//	Function: ExtendLPIfPossible()
//	Description: Helper function
//				 Pass in a device that is controlled byt a SV - extend at low pressure if possible
//	Created by: Ben Hess
//	Created Date: June 27th, 2019

IF (__QUERYINTERFACE(device, extendLowPressureDevice)) THEN
	extendLowPressureDevice.ExtendLowPressure();
	ExtendLPIfPossible := TRUE;
ELSE
	ExtendLPIfPossible := FALSE;
END_IF

END_FUNCTION

// Testing/HelperFunctions/HomeIfNeeded
FUNCTION HomeIfNeeded : BOOL
VAR_INPUT
	Component : IComponent;
END_VAR
VAR
	homableDevice : IHomable;
END_VAR

//	Function: HomeIfNeeded()
//	Description: Helper function
//				 Pass in a component - if it has a homable motor, and is not yet homed, start homing
//	Created by: Ben Hess
//	Created Date: May 16th, 2019

IF (__QUERYINTERFACE(Component, homableDevice)) AND Component.OptionActive THEN
	IF homableDevice.IsHomed THEN
		HomeIfNeeded := TRUE;
		RETURN;
	ELSE
		homableDevice.HomeNow();
	END_IF
END_IF

END_FUNCTION

// Testing/HelperFunctions/MoveRequested
FUNCTION MoveRequested : BOOL
VAR_INPUT
	Component : IComponent;
END_VAR
VAR
	movableDevice : IPostHomeMove;
END_VAR

//	Function: MoveIfNeeded()
//	Description: Helper function
//				 Pass in a component - if it has a homable motor, and is not yet homed, start homing
//	Created by: Ben Hess
//	Created Date: May 16th, 2019

IF (__QUERYINTERFACE(Component, movableDevice)) AND Component.OptionActive THEN
	IF NOT movableDevice.InDesiredPosition THEN
		MoveRequested := TRUE;
		RETURN;
	ELSE
		RETURN;
	END_IF
END_IF

END_FUNCTION

// Testing/Motors/IPostHomeMove
INTERFACE IPostHomeMove

END_INTERFACE

// Testing/HelperFunctions/PostHomeMoveIfNeeded
FUNCTION PostHomeMoveIfNeeded : BOOL
VAR_INPUT
	Component : IComponent;
END_VAR
VAR
	movableDevice : IPostHomeMove;
END_VAR

//	Function: MoveIfNeeded()
//	Description: Helper function
//				 Pass in a component - if it has a homable motor, and is homed, and is configured for a post homing move, perform it
//	Created by: Ben Hess
//	Created Date: May 16th, 2019

IF (__QUERYINTERFACE(Component, movableDevice)) AND Component.OptionActive THEN
	IF movableDevice.InDesiredPosition THEN
		PostHomeMoveIfNeeded := TRUE;
		RETURN;
	ELSE
		movableDevice.MoveNow();
	END_IF
END_IF

END_FUNCTION

// Testing/Motors/FB_AppliedMotionMotor
FUNCTION_BLOCK FB_AppliedMotionMotor EXTENDS Axis_REF
VAR_INPUT
END_VAR
VAR_OUTPUT
END_VAR
VAR
END_VAR

END_FUNCTION_BLOCK

// UN00 - Sharp Bagger/EM01 - Bagger Head/TestBaggerHead
PROGRAM TestBaggerHead
VAR
END_VAR

END_PROGRAM

// /VISU_HELPER_Combobox_BagOpenFingersSelection
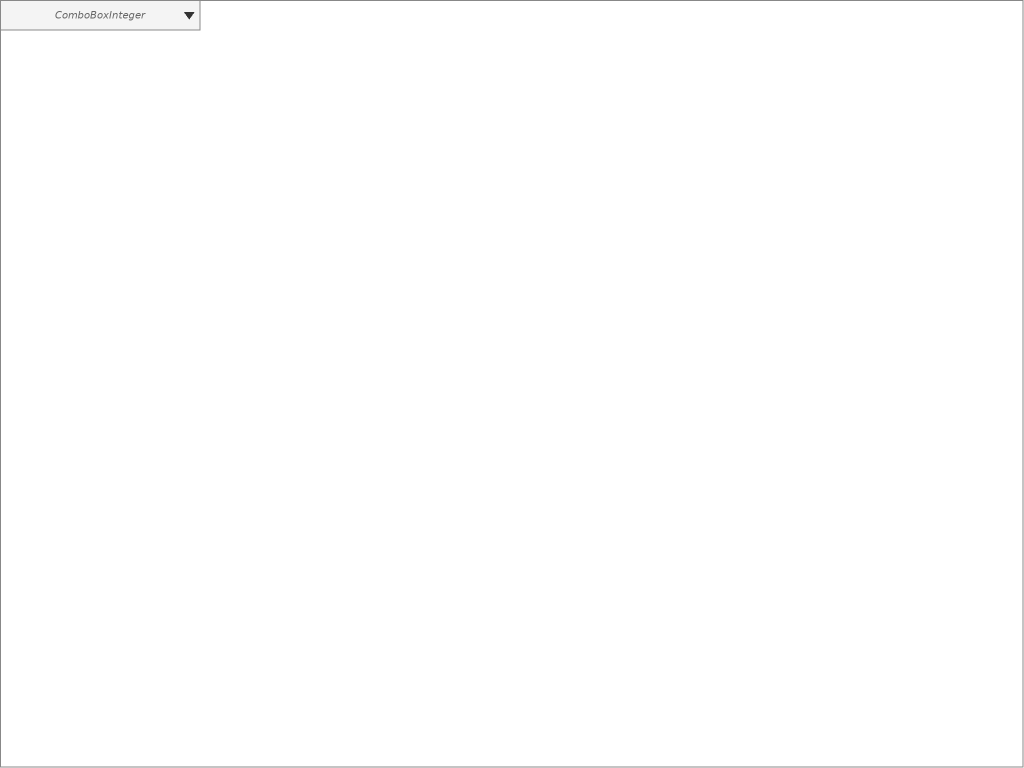
VISUALIZATION VISU_HELPER_Combobox_BagOpenFingersSelection  // 1024x768
VAR_IN_OUT
    varEnum : BagOpenFingersSelection;
END_VAR
    ComboBoxInteger (0,0 200x30), variable: varEnum, text list: 'TextListForCombobox_BagOpenFingersSelection'
END_VISUALIZATION

// /VISU_HELPER_Combobox_IntegratedConveyorSelection
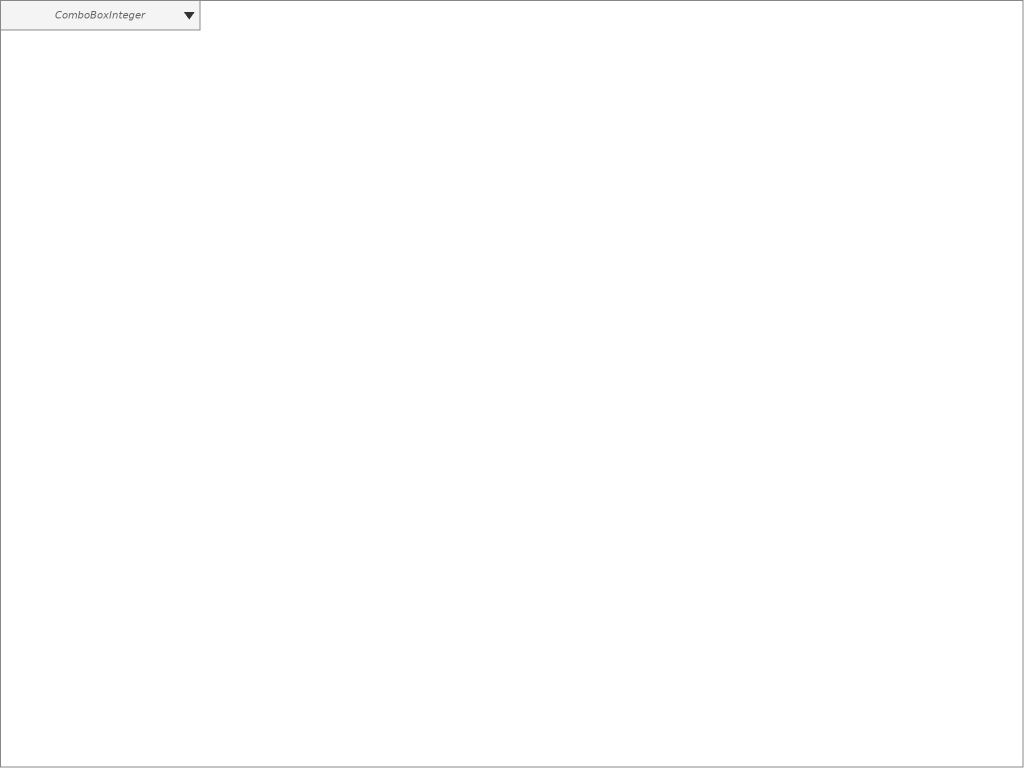
VISUALIZATION VISU_HELPER_Combobox_IntegratedConveyorSelection  // 1024x768
VAR_IN_OUT
    varEnum : IntegratedConveyorSelection;
END_VAR
    ComboBoxInteger (0,0 200x30), variable: varEnum, text list: 'TextListForCombobox_IntegratedConveyorSelection'
END_VISUALIZATION

// /VISU_HELPER_Combobox_LabelPrinterSelection
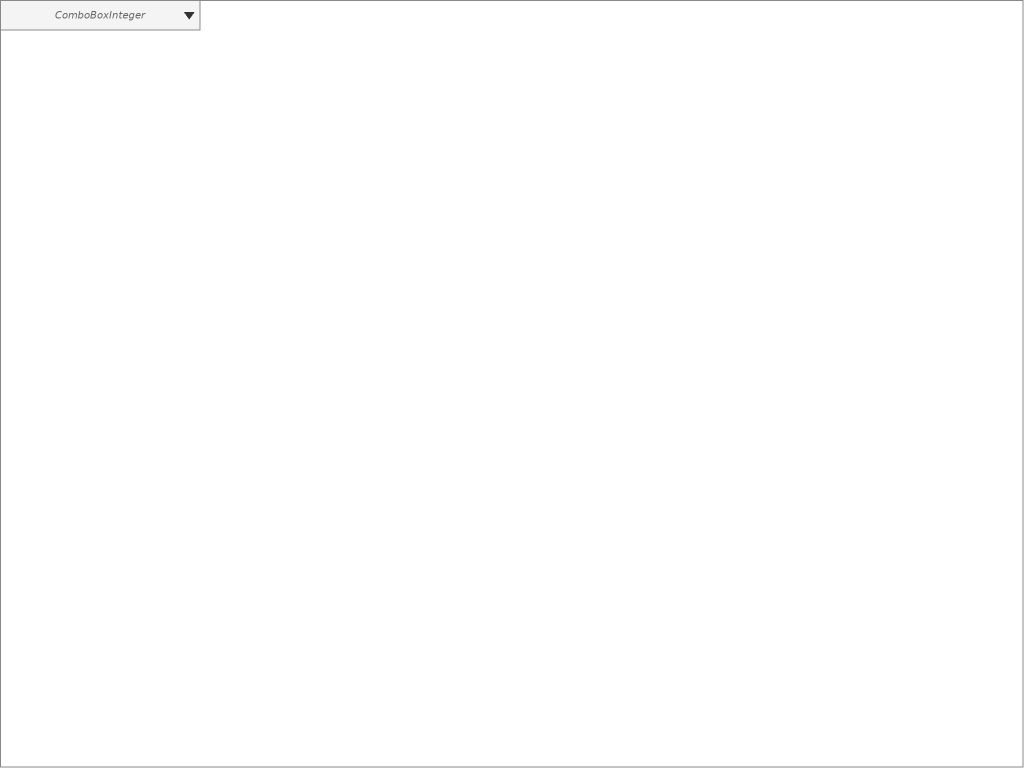
VISUALIZATION VISU_HELPER_Combobox_LabelPrinterSelection  // 1024x768
VAR_IN_OUT
    varEnum : LabelPrinterSelection;
END_VAR
    ComboBoxInteger (0,0 200x30), variable: varEnum, text list: 'TextListForCombobox_LabelPrinterSelection'
END_VISUALIZATION

// /VISU_HELPER_Combobox_PackageEjectionSelection
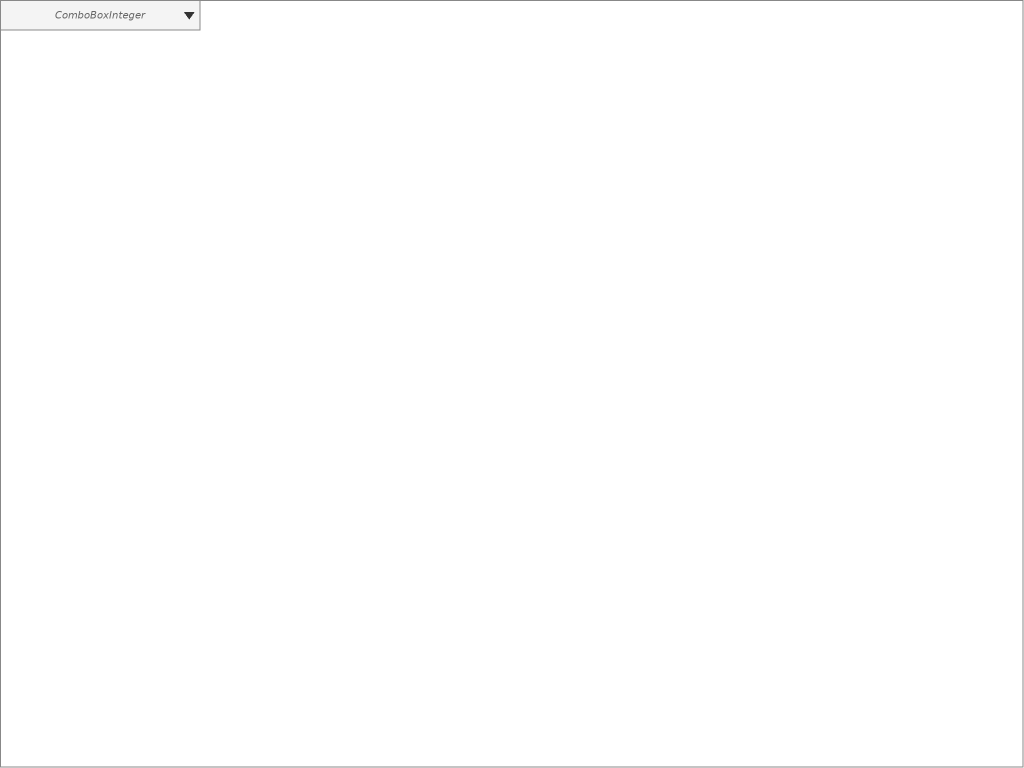
VISUALIZATION VISU_HELPER_Combobox_PackageEjectionSelection  // 1024x768
VAR_IN_OUT
    varEnum : PackageEjectionSelection;
END_VAR
    ComboBoxInteger (0,0 200x30), variable: varEnum, text list: 'TextListForCombobox_PackageEjectionSelection'
END_VISUALIZATION

// /VISU_HELPER_Combobox_SealFlattenerSelection
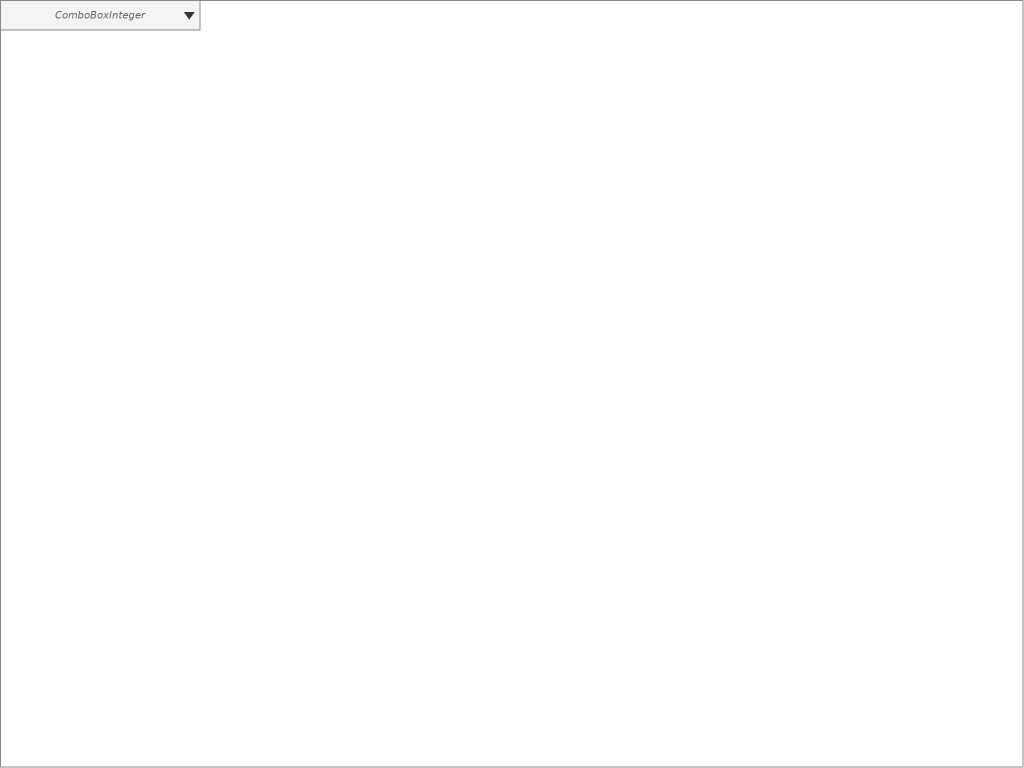
VISUALIZATION VISU_HELPER_Combobox_SealFlattenerSelection  // 1024x768
VAR_IN_OUT
    varEnum : SealFlattenerSelection;
END_VAR
    ComboBoxInteger (0,0 200x30), variable: varEnum, text list: 'TextListForCombobox_SealFlattenerSelection'
END_VISUALIZATION

// /VISU_NEW_FB_HMIData
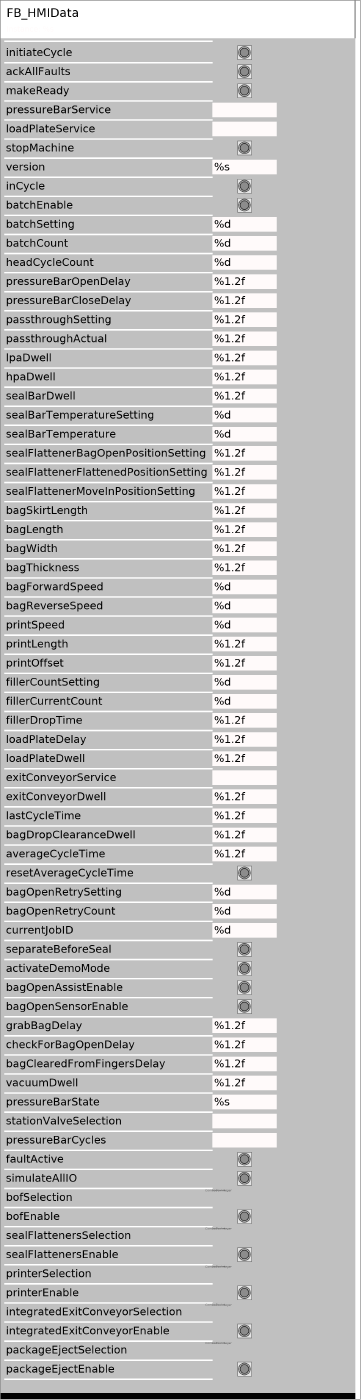
VISUALIZATION VISU_NEW_FB_HMIData  // 607x2348
VAR_INPUT
   {attribute 'parameterstringof' := 'm_Input_FB'}
   m_Input_INST_Str : STRING;
END_VAR
VAR_IN_OUT
   m_Input_FB : FB_HMIData;
END_VAR
    RoundedRectangle (0,0 597x81)
    RoundedRectangle (0,2306 597x40)
    Rectangle (0,64 597x2272)
    PushSwitch (399,76 24x24), variable: m_Input_FB.initiateCycle, behaviour: TOGGLE, style: Switch-PushSwitch-Gray
    PushSwitch (399,108 24x24), variable: m_Input_FB.ackAllFaults, behaviour: TOGGLE, style: Switch-PushSwitch-Gray
    PushSwitch (399,140 24x24), variable: m_Input_FB.makeReady, behaviour: TOGGLE, style: Switch-PushSwitch-Gray
    PushSwitch (399,236 24x24), variable: m_Input_FB.stopMachine, behaviour: TOGGLE, style: Switch-PushSwitch-Gray
    PushSwitch (399,300 24x24), variable: m_Input_FB.inCycle, behaviour: TOGGLE, style: Switch-PushSwitch-Gray
    PushSwitch (399,332 24x24), variable: m_Input_FB.batchEnable, behaviour: TOGGLE, style: Switch-PushSwitch-Gray
    PushSwitch (399,1452 24x24), variable: m_Input_FB.resetAverageCycleTime, behaviour: TOGGLE, style: Switch-PushSwitch-Gray
    PushSwitch (399,1580 24x24), variable: m_Input_FB.separateBeforeSeal, behaviour: TOGGLE, style: Switch-PushSwitch-Gray
    PushSwitch (399,1612 24x24), variable: m_Input_FB.activateDemoMode, behaviour: TOGGLE, style: Switch-PushSwitch-Gray
    PushSwitch (399,1644 24x24), variable: m_Input_FB.bagOpenAssistEnable, behaviour: TOGGLE, style: Switch-PushSwitch-Gray
    PushSwitch (399,1676 24x24), variable: m_Input_FB.bagOpenSensorEnable, behaviour: TOGGLE, style: Switch-PushSwitch-Gray
    PushSwitch (399,1932 24x24), variable: m_Input_FB.faultActive, behaviour: TOGGLE, style: Switch-PushSwitch-Gray
    PushSwitch (399,1964 24x24), variable: m_Input_FB.simulateAllIO, behaviour: TOGGLE, style: Switch-PushSwitch-Gray
    PushSwitch (399,2028 24x24), variable: m_Input_FB.bofEnable, behaviour: TOGGLE, style: Switch-PushSwitch-Gray
    PushSwitch (399,2092 24x24), variable: m_Input_FB.sealFlattenersEnable, behaviour: TOGGLE, style: Switch-PushSwitch-Gray
    PushSwitch (399,2156 24x24), variable: m_Input_FB.printerEnable, behaviour: TOGGLE, style: Switch-PushSwitch-Gray
    PushSwitch (399,2220 24x24), variable: m_Input_FB.integratedExitConveyorEnable, behaviour: TOGGLE, style: Switch-PushSwitch-Gray
    PushSwitch (399,2284 24x24), variable: m_Input_FB.packageEjectEnable, behaviour: TOGGLE, style: Switch-PushSwitch-Gray
    Rectangle (8,8 597x27), "FB_HMIData"
    Rectangle (8,35 597x27), "Instance: %s", text variable: m_Input_INST_Str
    Rectangle (7,68 350x2)
    Rectangle (7,76 350x24), "initiateCycle"
    Rectangle (7,104 350x2)
    Rectangle (7,108 350x24), "ackAllFaults"
    Rectangle (7,136 350x2)
    Rectangle (7,140 350x24), "makeReady"
    Rectangle (7,168 350x2)
    Rectangle (357,172 108x24), text variable: m_Input_FB.pressureBarService
        OnMouseClick: write the text variable via Default
    Rectangle (7,172 350x24), "pressureBarService"
    Rectangle (7,200 350x2)
    Rectangle (357,204 108x24), text variable: m_Input_FB.loadPlateService
        OnMouseClick: write the text variable via Default
    Rectangle (7,204 350x24), "loadPlateService"
    Rectangle (7,232 350x2)
    Rectangle (7,236 350x24), "stopMachine"
    Rectangle (7,264 350x2)
    Rectangle (357,268 108x24), "%s", text variable: m_Input_FB.version
        OnMouseClick: write the text variable via Default
    Rectangle (7,268 350x24), "version"
    Rectangle (7,296 350x2)
    Rectangle (7,300 350x24), "inCycle"
    Rectangle (7,328 350x2)
    Rectangle (7,332 350x24), "batchEnable"
    Rectangle (7,360 350x2)
    Rectangle (357,364 108x24), "%d", text variable: m_Input_FB.batchSetting
        OnMouseClick: write the text variable via Default
    Rectangle (7,364 350x24), "batchSetting"
    Rectangle (7,392 350x2)
    Rectangle (357,396 108x24), "%d", text variable: m_Input_FB.batchCount
        OnMouseClick: write the text variable via Default
    Rectangle (7,396 350x24), "batchCount"
    Rectangle (7,424 350x2)
    Rectangle (357,428 108x24), "%d", text variable: m_Input_FB.headCycleCount
        OnMouseClick: write the text variable via Default
    Rectangle (7,428 350x24), "headCycleCount"
    Rectangle (7,456 350x2)
    Rectangle (357,460 108x24), "%1.2f", text variable: m_Input_FB.pressureBarOpenDelay
        OnMouseClick: write the text variable via Default
    Rectangle (7,460 350x24), "pressureBarOpenDelay"
    Rectangle (7,488 350x2)
    Rectangle (357,492 108x24), "%1.2f", text variable: m_Input_FB.pressureBarCloseDelay
        OnMouseClick: write the text variable via Default
    Rectangle (7,492 350x24), "pressureBarCloseDelay"
    Rectangle (7,520 350x2)
    Rectangle (357,524 108x24), "%1.2f", text variable: m_Input_FB.passthroughSetting
        OnMouseClick: write the text variable via Default
    Rectangle (7,524 350x24), "passthroughSetting"
    Rectangle (7,552 350x2)
    Rectangle (357,556 108x24), "%1.2f", text variable: m_Input_FB.passthroughActual
        OnMouseClick: write the text variable via Default
    Rectangle (7,556 350x24), "passthroughActual"
    Rectangle (7,584 350x2)
    Rectangle (357,588 108x24), "%1.2f", text variable: m_Input_FB.lpaDwell
        OnMouseClick: write the text variable via Default
    Rectangle (7,588 350x24), "lpaDwell"
    Rectangle (7,616 350x2)
    Rectangle (357,620 108x24), "%1.2f", text variable: m_Input_FB.hpaDwell
        OnMouseClick: write the text variable via Default
    Rectangle (7,620 350x24), "hpaDwell"
    Rectangle (7,648 350x2)
    Rectangle (357,652 108x24), "%1.2f", text variable: m_Input_FB.sealBarDwell
        OnMouseClick: write the text variable via Default
    Rectangle (7,652 350x24), "sealBarDwell"
    Rectangle (7,680 350x2)
    Rectangle (357,684 108x24), "%d", text variable: m_Input_FB.sealBarTemperatureSetting
        OnMouseClick: write the text variable via Default
    Rectangle (7,684 350x24), "sealBarTemperatureSetting"
    Rectangle (7,712 350x2)
    Rectangle (357,716 108x24), "%d", text variable: m_Input_FB.sealBarTemperature
        OnMouseClick: write the text variable via Default
    Rectangle (7,716 350x24), "sealBarTemperature"
    Rectangle (7,744 350x2)
    Rectangle (357,748 108x24), "%1.2f", text variable: m_Input_FB.sealFlattenerBagOpenPositionSetting
        OnMouseClick: write the text variable via Default
    Rectangle (7,748 350x24), "sealFlattenerBagOpenPositionSetting"
    Rectangle (7,776 350x2)
    Rectangle (357,780 108x24), "%1.2f", text variable: m_Input_FB.sealFlattenerFlattenedPositionSetting
        OnMouseClick: write the text variable via Default
    Rectangle (7,780 350x24), "sealFlattenerFlattenedPositionSetting"
    Rectangle (7,808 350x2)
    Rectangle (357,812 108x24), "%1.2f", text variable: m_Input_FB.sealFlattenerMoveInPositionSetting
        OnMouseClick: write the text variable via Default
    Rectangle (7,812 350x24), "sealFlattenerMoveInPositionSetting"
    Rectangle (7,840 350x2)
    Rectangle (357,844 108x24), "%1.2f", text variable: m_Input_FB.bagSkirtLength
        OnMouseClick: write the text variable via Default
    Rectangle (7,844 350x24), "bagSkirtLength"
    Rectangle (7,872 350x2)
    Rectangle (357,876 108x24), "%1.2f", text variable: m_Input_FB.bagLength
        OnMouseClick: write the text variable via Default
    Rectangle (7,876 350x24), "bagLength"
    Rectangle (7,904 350x2)
    Rectangle (357,908 108x24), "%1.2f", text variable: m_Input_FB.bagWidth
        OnMouseClick: write the text variable via Default
    Rectangle (7,908 350x24), "bagWidth"
    Rectangle (7,936 350x2)
    Rectangle (357,940 108x24), "%1.2f", text variable: m_Input_FB.bagThickness
        OnMouseClick: write the text variable via Default
    Rectangle (7,940 350x24), "bagThickness"
    Rectangle (7,968 350x2)
    Rectangle (357,972 108x24), "%d", text variable: m_Input_FB.bagForwardSpeed
        OnMouseClick: write the text variable via Default
    Rectangle (7,972 350x24), "bagForwardSpeed"
    Rectangle (7,1000 350x2)
    Rectangle (357,1004 108x24), "%d", text variable: m_Input_FB.bagReverseSpeed
        OnMouseClick: write the text variable via Default
    Rectangle (7,1004 350x24), "bagReverseSpeed"
    Rectangle (7,1032 350x2)
    Rectangle (357,1036 108x24), "%d", text variable: m_Input_FB.printSpeed
        OnMouseClick: write the text variable via Default
    Rectangle (7,1036 350x24), "printSpeed"
    Rectangle (7,1064 350x2)
    Rectangle (357,1068 108x24), "%1.2f", text variable: m_Input_FB.printLength
        OnMouseClick: write the text variable via Default
    Rectangle (7,1068 350x24), "printLength"
    Rectangle (7,1096 350x2)
    Rectangle (357,1100 108x24), "%1.2f", text variable: m_Input_FB.printOffset
        OnMouseClick: write the text variable via Default
    Rectangle (7,1100 350x24), "printOffset"
    Rectangle (7,1128 350x2)
    Rectangle (357,1132 108x24), "%d", text variable: m_Input_FB.fillerCountSetting
        OnMouseClick: write the text variable via Default
    Rectangle (7,1132 350x24), "fillerCountSetting"
    Rectangle (7,1160 350x2)
    Rectangle (357,1164 108x24), "%d", text variable: m_Input_FB.fillerCurrentCount
        OnMouseClick: write the text variable via Default
    Rectangle (7,1164 350x24), "fillerCurrentCount"
    Rectangle (7,1192 350x2)
    Rectangle (357,1196 108x24), "%1.2f", text variable: m_Input_FB.fillerDropTime
        OnMouseClick: write the text variable via Default
    Rectangle (7,1196 350x24), "fillerDropTime"
    Rectangle (7,1224 350x2)
    Rectangle (357,1228 108x24), "%1.2f", text variable: m_Input_FB.loadPlateDelay
        OnMouseClick: write the text variable via Default
    Rectangle (7,1228 350x24), "loadPlateDelay"
    Rectangle (7,1256 350x2)
    Rectangle (357,1260 108x24), "%1.2f", text variable: m_Input_FB.loadPlateDwell
        OnMouseClick: write the text variable via Default
    Rectangle (7,1260 350x24), "loadPlateDwell"
    Rectangle (7,1288 350x2)
    Rectangle (357,1292 108x24), text variable: m_Input_FB.exitConveyorService
        OnMouseClick: write the text variable via Default
    Rectangle (7,1292 350x24), "exitConveyorService"
    Rectangle (7,1320 350x2)
    Rectangle (357,1324 108x24), "%1.2f", text variable: m_Input_FB.exitConveyorDwell
        OnMouseClick: write the text variable via Default
    Rectangle (7,1324 350x24), "exitConveyorDwell"
    Rectangle (7,1352 350x2)
    Rectangle (357,1356 108x24), "%1.2f", text variable: m_Input_FB.lastCycleTime
        OnMouseClick: write the text variable via Default
    Rectangle (7,1356 350x24), "lastCycleTime"
    Rectangle (7,1384 350x2)
    Rectangle (357,1388 108x24), "%1.2f", text variable: m_Input_FB.bagDropClearanceDwell
        OnMouseClick: write the text variable via Default
    Rectangle (7,1388 350x24), "bagDropClearanceDwell"
    Rectangle (7,1416 350x2)
    Rectangle (357,1420 108x24), "%1.2f", text variable: m_Input_FB.averageCycleTime
        OnMouseClick: write the text variable via Default
    Rectangle (7,1420 350x24), "averageCycleTime"
    Rectangle (7,1448 350x2)
    Rectangle (7,1452 350x24), "resetAverageCycleTime"
    Rectangle (7,1480 350x2)
    Rectangle (357,1484 108x24), "%d", text variable: m_Input_FB.bagOpenRetrySetting
        OnMouseClick: write the text variable via Default
    Rectangle (7,1484 350x24), "bagOpenRetrySetting"
    Rectangle (7,1512 350x2)
    Rectangle (357,1516 108x24), "%d", text variable: m_Input_FB.bagOpenRetryCount
        OnMouseClick: write the text variable via Default
    Rectangle (7,1516 350x24), "bagOpenRetryCount"
    Rectangle (7,1544 350x2)
    Rectangle (357,1548 108x24), "%d", text variable: m_Input_FB.currentJobID
        OnMouseClick: write the text variable via Default
    Rectangle (7,1548 350x24), "currentJobID"
    Rectangle (7,1576 350x2)
    Rectangle (7,1580 350x24), "separateBeforeSeal"
    Rectangle (7,1608 350x2)
    Rectangle (7,1612 350x24), "activateDemoMode"
    Rectangle (7,1640 350x2)
    Rectangle (7,1644 350x24), "bagOpenAssistEnable"
    Rectangle (7,1672 350x2)
    Rectangle (7,1676 350x24), "bagOpenSensorEnable"
    Rectangle (7,1704 350x2)
    Rectangle (357,1708 108x24), "%1.2f", text variable: m_Input_FB.grabBagDelay
        OnMouseClick: write the text variable via Default
    Rectangle (7,1708 350x24), "grabBagDelay"
    Rectangle (7,1736 350x2)
    Rectangle (357,1740 108x24), "%1.2f", text variable: m_Input_FB.checkForBagOpenDelay
        OnMouseClick: write the text variable via Default
    Rectangle (7,1740 350x24), "checkForBagOpenDelay"
    Rectangle (7,1768 350x2)
    Rectangle (357,1772 108x24), "%1.2f", text variable: m_Input_FB.bagClearedFromFingersDelay
        OnMouseClick: write the text variable via Default
    Rectangle (7,1772 350x24), "bagClearedFromFingersDelay"
    Rectangle (7,1800 350x2)
    Rectangle (357,1804 108x24), "%1.2f", text variable: m_Input_FB.vacuumDwell
        OnMouseClick: write the text variable via Default
    Rectangle (7,1804 350x24), "vacuumDwell"
    Rectangle (7,1832 350x2)
    Rectangle (357,1836 108x24), "%s", text variable: m_Input_FB.pressureBarState
        OnMouseClick: write the text variable via Default
    Rectangle (7,1836 350x24), "pressureBarState"
    Rectangle (7,1864 350x2)
    Rectangle (357,1868 108x24), text variable: m_Input_FB.stationValveSelection
        OnMouseClick: write the text variable via Default
    Rectangle (7,1868 350x24), "stationValveSelection"
    Rectangle (7,1896 350x2)
    Rectangle (357,1900 108x24), text variable: m_Input_FB.pressureBarCycles
        OnMouseClick: write the text variable via Default
    Rectangle (7,1900 350x24), "pressureBarCycles"
    Rectangle (7,1928 350x2)
    Rectangle (7,1932 350x24), "faultActive"
    Rectangle (7,1960 350x2)
    Rectangle (7,1964 350x24), "simulateAllIO"
    Rectangle (7,1992 350x2)
    Rectangle (7,1996 350x24), "bofSelection"
    Rectangle (7,2024 350x2)
    Rectangle (7,2028 350x24), "bofEnable"
    Rectangle (7,2056 350x2)
    Rectangle (7,2060 350x24), "sealFlattenersSelection"
    Rectangle (7,2088 350x2)
    Rectangle (7,2092 350x24), "sealFlattenersEnable"
    Rectangle (7,2120 350x2)
    Rectangle (7,2124 350x24), "printerSelection"
    Rectangle (7,2152 350x2)
    Rectangle (7,2156 350x24), "printerEnable"
    Rectangle (7,2184 350x2)
    Rectangle (7,2188 350x24), "integratedExitConveyorSelection"
    Rectangle (7,2216 350x2)
    Rectangle (7,2220 350x24), "integratedExitConveyorEnable"
    Rectangle (7,2248 350x2)
    Rectangle (7,2252 350x24), "packageEjectSelection"
    Rectangle (7,2280 350x2)
    Rectangle (7,2284 350x24), "packageEjectEnable"
    Rectangle (7,2312 350x2)
    Frame (357,1996 108x24)
        shows VISU_HELPER_Combobox_BagOpenFingersSelection(varEnum := m_Input_FB.bofSelection)
    Frame (357,2060 108x24)
        shows VISU_HELPER_Combobox_SealFlattenerSelection(varEnum := m_Input_FB.sealFlattenersSelection)
    Frame (357,2124 108x24)
        shows VISU_HELPER_Combobox_LabelPrinterSelection(varEnum := m_Input_FB.printerSelection)
    Frame (357,2188 108x24)
        shows VISU_HELPER_Combobox_IntegratedConveyorSelection(varEnum := m_Input_FB.integratedExitConveyorSelection)
    Frame (357,2252 108x24)
        shows VISU_HELPER_Combobox_PackageEjectionSelection(varEnum := m_Input_FB.packageEjectSelection)
END_VISUALIZATION

// /VISU_NEW_FB_IOLinkBlock
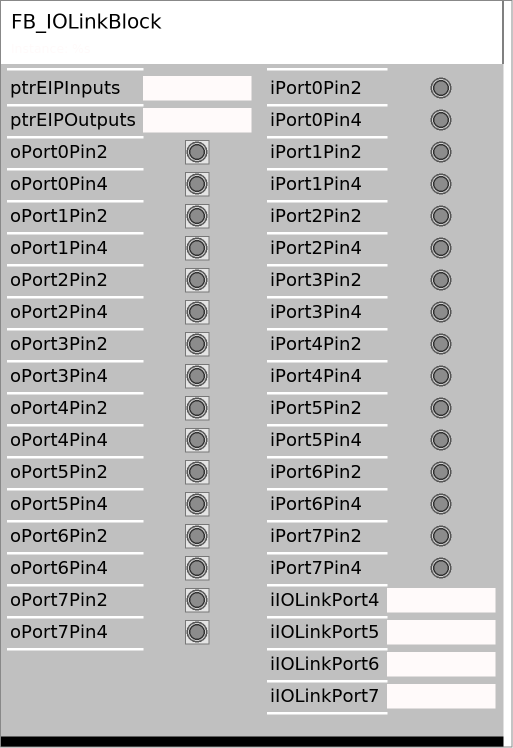
VISUALIZATION VISU_NEW_FB_IOLinkBlock  // 513x748
VAR_INPUT
   {attribute 'parameterstringof' := 'm_Input_FB'}
   m_Input_INST_Str : STRING;
END_VAR
VAR_IN_OUT
   m_Input_FB : FB_IOLinkBlock;
END_VAR
    RoundedRectangle (0,0 503x81)
    RoundedRectangle (0,706 503x40)
    Rectangle (0,64 503x672)
    Lamp1 (429,76 24x24), variable: m_Input_FB.iPort0Pin2, style: Lamp-Lamp1-Gray
    Lamp1 (429,108 24x24), variable: m_Input_FB.iPort0Pin4, style: Lamp-Lamp1-Gray
    Lamp1 (429,140 24x24), variable: m_Input_FB.iPort1Pin2, style: Lamp-Lamp1-Gray
    Lamp1 (429,172 24x24), variable: m_Input_FB.iPort1Pin4, style: Lamp-Lamp1-Gray
    Lamp1 (429,204 24x24), variable: m_Input_FB.iPort2Pin2, style: Lamp-Lamp1-Gray
    Lamp1 (429,236 24x24), variable: m_Input_FB.iPort2Pin4, style: Lamp-Lamp1-Gray
    Lamp1 (429,268 24x24), variable: m_Input_FB.iPort3Pin2, style: Lamp-Lamp1-Gray
    Lamp1 (429,300 24x24), variable: m_Input_FB.iPort3Pin4, style: Lamp-Lamp1-Gray
    Lamp1 (429,332 24x24), variable: m_Input_FB.iPort4Pin2, style: Lamp-Lamp1-Gray
    Lamp1 (429,364 24x24), variable: m_Input_FB.iPort4Pin4, style: Lamp-Lamp1-Gray
    Lamp1 (429,396 24x24), variable: m_Input_FB.iPort5Pin2, style: Lamp-Lamp1-Gray
    Lamp1 (429,428 24x24), variable: m_Input_FB.iPort5Pin4, style: Lamp-Lamp1-Gray
    Lamp1 (429,460 24x24), variable: m_Input_FB.iPort6Pin2, style: Lamp-Lamp1-Gray
    Lamp1 (429,492 24x24), variable: m_Input_FB.iPort6Pin4, style: Lamp-Lamp1-Gray
    Lamp1 (429,524 24x24), variable: m_Input_FB.iPort7Pin2, style: Lamp-Lamp1-Gray
    Lamp1 (429,556 24x24), variable: m_Input_FB.iPort7Pin4, style: Lamp-Lamp1-Gray
    PushSwitch (185,140 24x24), variable: m_Input_FB.oPort0Pin2, behaviour: TOGGLE, style: Switch-PushSwitch-Gray
    PushSwitch (185,172 24x24), variable: m_Input_FB.oPort0Pin4, behaviour: TOGGLE, style: Switch-PushSwitch-Gray
    PushSwitch (185,204 24x24), variable: m_Input_FB.oPort1Pin2, behaviour: TOGGLE, style: Switch-PushSwitch-Gray
    PushSwitch (185,236 24x24), variable: m_Input_FB.oPort1Pin4, behaviour: TOGGLE, style: Switch-PushSwitch-Gray
    PushSwitch (185,268 24x24), variable: m_Input_FB.oPort2Pin2, behaviour: TOGGLE, style: Switch-PushSwitch-Gray
    PushSwitch (185,300 24x24), variable: m_Input_FB.oPort2Pin4, behaviour: TOGGLE, style: Switch-PushSwitch-Gray
    PushSwitch (185,332 24x24), variable: m_Input_FB.oPort3Pin2, behaviour: TOGGLE, style: Switch-PushSwitch-Gray
    PushSwitch (185,364 24x24), variable: m_Input_FB.oPort3Pin4, behaviour: TOGGLE, style: Switch-PushSwitch-Gray
    PushSwitch (185,396 24x24), variable: m_Input_FB.oPort4Pin2, behaviour: TOGGLE, style: Switch-PushSwitch-Gray
    PushSwitch (185,428 24x24), variable: m_Input_FB.oPort4Pin4, behaviour: TOGGLE, style: Switch-PushSwitch-Gray
    PushSwitch (185,460 24x24), variable: m_Input_FB.oPort5Pin2, behaviour: TOGGLE, style: Switch-PushSwitch-Gray
    PushSwitch (185,492 24x24), variable: m_Input_FB.oPort5Pin4, behaviour: TOGGLE, style: Switch-PushSwitch-Gray
    PushSwitch (185,524 24x24), variable: m_Input_FB.oPort6Pin2, behaviour: TOGGLE, style: Switch-PushSwitch-Gray
    PushSwitch (185,556 24x24), variable: m_Input_FB.oPort6Pin4, behaviour: TOGGLE, style: Switch-PushSwitch-Gray
    PushSwitch (185,588 24x24), variable: m_Input_FB.oPort7Pin2, behaviour: TOGGLE, style: Switch-PushSwitch-Gray
    PushSwitch (185,620 24x24), variable: m_Input_FB.oPort7Pin4, behaviour: TOGGLE, style: Switch-PushSwitch-Gray
    Rectangle (8,8 503x27), "FB_IOLinkBlock"
    Rectangle (8,35 503x27), "Instance: %s", text variable: m_Input_INST_Str
    Rectangle (7,68 136x2)
    Rectangle (143,76 108x24), text variable: m_Input_FB.ptrEIPInputs
        OnMouseClick: write the text variable via Default
    Rectangle (7,76 136x24), "ptrEIPInputs"
    Rectangle (7,104 136x2)
    Rectangle (143,108 108x24), text variable: m_Input_FB.ptrEIPOutputs
        OnMouseClick: write the text variable via Default
    Rectangle (7,108 136x24), "ptrEIPOutputs"
    Rectangle (7,136 136x2)
    Rectangle (7,140 136x24), "oPort0Pin2"
    Rectangle (7,168 136x2)
    Rectangle (7,172 136x24), "oPort0Pin4"
    Rectangle (7,200 136x2)
    Rectangle (7,204 136x24), "oPort1Pin2"
    Rectangle (7,232 136x2)
    Rectangle (7,236 136x24), "oPort1Pin4"
    Rectangle (7,264 136x2)
    Rectangle (7,268 136x24), "oPort2Pin2"
    Rectangle (7,296 136x2)
    Rectangle (7,300 136x24), "oPort2Pin4"
    Rectangle (7,328 136x2)
    Rectangle (7,332 136x24), "oPort3Pin2"
    Rectangle (7,360 136x2)
    Rectangle (7,364 136x24), "oPort3Pin4"
    Rectangle (7,392 136x2)
    Rectangle (7,396 136x24), "oPort4Pin2"
    Rectangle (7,424 136x2)
    Rectangle (7,428 136x24), "oPort4Pin4"
    Rectangle (7,456 136x2)
    Rectangle (7,460 136x24), "oPort5Pin2"
    Rectangle (7,488 136x2)
    Rectangle (7,492 136x24), "oPort5Pin4"
    Rectangle (7,520 136x2)
    Rectangle (7,524 136x24), "oPort6Pin2"
    Rectangle (7,552 136x2)
    Rectangle (7,556 136x24), "oPort6Pin4"
    Rectangle (7,584 136x2)
    Rectangle (7,588 136x24), "oPort7Pin2"
    Rectangle (7,616 136x2)
    Rectangle (7,620 136x24), "oPort7Pin4"
    Rectangle (7,648 136x2)
    Rectangle (267,68 120x2)
    Rectangle (267,76 120x24), "iPort0Pin2"
    Rectangle (267,104 120x2)
    Rectangle (267,108 120x24), "iPort0Pin4"
    Rectangle (267,136 120x2)
    Rectangle (267,140 120x24), "iPort1Pin2"
    Rectangle (267,168 120x2)
    Rectangle (267,172 120x24), "iPort1Pin4"
    Rectangle (267,200 120x2)
    Rectangle (267,204 120x24), "iPort2Pin2"
    Rectangle (267,232 120x2)
    Rectangle (267,236 120x24), "iPort2Pin4"
    Rectangle (267,264 120x2)
    Rectangle (267,268 120x24), "iPort3Pin2"
    Rectangle (267,296 120x2)
    Rectangle (267,300 120x24), "iPort3Pin4"
    Rectangle (267,328 120x2)
    Rectangle (267,332 120x24), "iPort4Pin2"
    Rectangle (267,360 120x2)
    Rectangle (267,364 120x24), "iPort4Pin4"
    Rectangle (267,392 120x2)
    Rectangle (267,396 120x24), "iPort5Pin2"
    Rectangle (267,424 120x2)
    Rectangle (267,428 120x24), "iPort5Pin4"
    Rectangle (267,456 120x2)
    Rectangle (267,460 120x24), "iPort6Pin2"
    Rectangle (267,488 120x2)
    Rectangle (267,492 120x24), "iPort6Pin4"
    Rectangle (267,520 120x2)
    Rectangle (267,524 120x24), "iPort7Pin2"
    Rectangle (267,552 120x2)
    Rectangle (267,556 120x24), "iPort7Pin4"
    Rectangle (267,584 120x2)
    Rectangle (387,588 108x24), text variable: m_Input_FB.iIOLinkPort4
    Rectangle (267,588 120x24), "iIOLinkPort4"
    Rectangle (267,616 120x2)
    Rectangle (387,620 108x24), text variable: m_Input_FB.iIOLinkPort5
    Rectangle (267,620 120x24), "iIOLinkPort5"
    Rectangle (267,648 120x2)
    Rectangle (387,652 108x24), text variable: m_Input_FB.iIOLinkPort6
    Rectangle (267,652 120x24), "iIOLinkPort6"
    Rectangle (267,680 120x2)
    Rectangle (387,684 108x24), text variable: m_Input_FB.iIOLinkPort7
    Rectangle (267,684 120x24), "iIOLinkPort7"
    Rectangle (267,712 120x2)
END_VISUALIZATION

// /VISU_NEW_FB_Murr16PointCFGIO
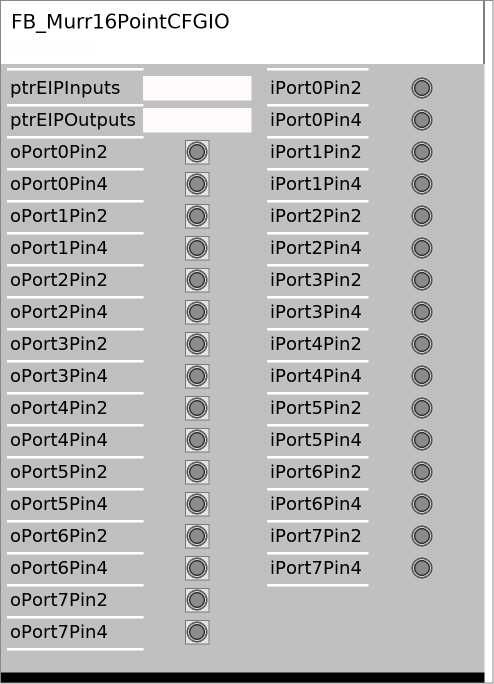
VISUALIZATION VISU_NEW_FB_Murr16PointCFGIO  // 494x684
VAR_INPUT
   {attribute 'parameterstringof' := 'm_Input_FB'}
   m_Input_INST_Str : STRING;
END_VAR
VAR_IN_OUT
   m_Input_FB : FB_Murr16PointCFGIO;
END_VAR
    RoundedRectangle (0,0 484x81)
    RoundedRectangle (0,642 484x40)
    Rectangle (0,64 484x608)
    Lamp1 (410,76 24x24), variable: m_Input_FB.iPort0Pin2, style: Lamp-Lamp1-Gray
    Lamp1 (410,108 24x24), variable: m_Input_FB.iPort0Pin4, style: Lamp-Lamp1-Gray
    Lamp1 (410,140 24x24), variable: m_Input_FB.iPort1Pin2, style: Lamp-Lamp1-Gray
    Lamp1 (410,172 24x24), variable: m_Input_FB.iPort1Pin4, style: Lamp-Lamp1-Gray
    Lamp1 (410,204 24x24), variable: m_Input_FB.iPort2Pin2, style: Lamp-Lamp1-Gray
    Lamp1 (410,236 24x24), variable: m_Input_FB.iPort2Pin4, style: Lamp-Lamp1-Gray
    Lamp1 (410,268 24x24), variable: m_Input_FB.iPort3Pin2, style: Lamp-Lamp1-Gray
    Lamp1 (410,300 24x24), variable: m_Input_FB.iPort3Pin4, style: Lamp-Lamp1-Gray
    Lamp1 (410,332 24x24), variable: m_Input_FB.iPort4Pin2, style: Lamp-Lamp1-Gray
    Lamp1 (410,364 24x24), variable: m_Input_FB.iPort4Pin4, style: Lamp-Lamp1-Gray
    Lamp1 (410,396 24x24), variable: m_Input_FB.iPort5Pin2, style: Lamp-Lamp1-Gray
    Lamp1 (410,428 24x24), variable: m_Input_FB.iPort5Pin4, style: Lamp-Lamp1-Gray
    Lamp1 (410,460 24x24), variable: m_Input_FB.iPort6Pin2, style: Lamp-Lamp1-Gray
    Lamp1 (410,492 24x24), variable: m_Input_FB.iPort6Pin4, style: Lamp-Lamp1-Gray
    Lamp1 (410,524 24x24), variable: m_Input_FB.iPort7Pin2, style: Lamp-Lamp1-Gray
    Lamp1 (410,556 24x24), variable: m_Input_FB.iPort7Pin4, style: Lamp-Lamp1-Gray
    PushSwitch (185,140 24x24), variable: m_Input_FB.oPort0Pin2, behaviour: TOGGLE, style: Switch-PushSwitch-Gray
    PushSwitch (185,172 24x24), variable: m_Input_FB.oPort0Pin4, behaviour: TOGGLE, style: Switch-PushSwitch-Gray
    PushSwitch (185,204 24x24), variable: m_Input_FB.oPort1Pin2, behaviour: TOGGLE, style: Switch-PushSwitch-Gray
    PushSwitch (185,236 24x24), variable: m_Input_FB.oPort1Pin4, behaviour: TOGGLE, style: Switch-PushSwitch-Gray
    PushSwitch (185,268 24x24), variable: m_Input_FB.oPort2Pin2, behaviour: TOGGLE, style: Switch-PushSwitch-Gray
    PushSwitch (185,300 24x24), variable: m_Input_FB.oPort2Pin4, behaviour: TOGGLE, style: Switch-PushSwitch-Gray
    PushSwitch (185,332 24x24), variable: m_Input_FB.oPort3Pin2, behaviour: TOGGLE, style: Switch-PushSwitch-Gray
    PushSwitch (185,364 24x24), variable: m_Input_FB.oPort3Pin4, behaviour: TOGGLE, style: Switch-PushSwitch-Gray
    PushSwitch (185,396 24x24), variable: m_Input_FB.oPort4Pin2, behaviour: TOGGLE, style: Switch-PushSwitch-Gray
    PushSwitch (185,428 24x24), variable: m_Input_FB.oPort4Pin4, behaviour: TOGGLE, style: Switch-PushSwitch-Gray
    PushSwitch (185,460 24x24), variable: m_Input_FB.oPort5Pin2, behaviour: TOGGLE, style: Switch-PushSwitch-Gray
    PushSwitch (185,492 24x24), variable: m_Input_FB.oPort5Pin4, behaviour: TOGGLE, style: Switch-PushSwitch-Gray
    PushSwitch (185,524 24x24), variable: m_Input_FB.oPort6Pin2, behaviour: TOGGLE, style: Switch-PushSwitch-Gray
    PushSwitch (185,556 24x24), variable: m_Input_FB.oPort6Pin4, behaviour: TOGGLE, style: Switch-PushSwitch-Gray
    PushSwitch (185,588 24x24), variable: m_Input_FB.oPort7Pin2, behaviour: TOGGLE, style: Switch-PushSwitch-Gray
    PushSwitch (185,620 24x24), variable: m_Input_FB.oPort7Pin4, behaviour: TOGGLE, style: Switch-PushSwitch-Gray
    Rectangle (8,8 484x27), "FB_Murr16PointCFGIO"
    Rectangle (8,35 484x27), "Instance: %s", text variable: m_Input_INST_Str
    Rectangle (7,68 136x2)
    Rectangle (143,76 108x24), text variable: m_Input_FB.ptrEIPInputs
        OnMouseClick: write the text variable via Default
    Rectangle (7,76 136x24), "ptrEIPInputs"
    Rectangle (7,104 136x2)
    Rectangle (143,108 108x24), text variable: m_Input_FB.ptrEIPOutputs
        OnMouseClick: write the text variable via Default
    Rectangle (7,108 136x24), "ptrEIPOutputs"
    Rectangle (7,136 136x2)
    Rectangle (7,140 136x24), "oPort0Pin2"
    Rectangle (7,168 136x2)
    Rectangle (7,172 136x24), "oPort0Pin4"
    Rectangle (7,200 136x2)
    Rectangle (7,204 136x24), "oPort1Pin2"
    Rectangle (7,232 136x2)
    Rectangle (7,236 136x24), "oPort1Pin4"
    Rectangle (7,264 136x2)
    Rectangle (7,268 136x24), "oPort2Pin2"
    Rectangle (7,296 136x2)
    Rectangle (7,300 136x24), "oPort2Pin4"
    Rectangle (7,328 136x2)
    Rectangle (7,332 136x24), "oPort3Pin2"
    Rectangle (7,360 136x2)
    Rectangle (7,364 136x24), "oPort3Pin4"
    Rectangle (7,392 136x2)
    Rectangle (7,396 136x24), "oPort4Pin2"
    Rectangle (7,424 136x2)
    Rectangle (7,428 136x24), "oPort4Pin4"
    Rectangle (7,456 136x2)
    Rectangle (7,460 136x24), "oPort5Pin2"
    Rectangle (7,488 136x2)
    Rectangle (7,492 136x24), "oPort5Pin4"
    Rectangle (7,520 136x2)
    Rectangle (7,524 136x24), "oPort6Pin2"
    Rectangle (7,552 136x2)
    Rectangle (7,556 136x24), "oPort6Pin4"
    Rectangle (7,584 136x2)
    Rectangle (7,588 136x24), "oPort7Pin2"
    Rectangle (7,616 136x2)
    Rectangle (7,620 136x24), "oPort7Pin4"
    Rectangle (7,648 136x2)
    Rectangle (267,68 101x2)
    Rectangle (267,76 101x24), "iPort0Pin2"
    Rectangle (267,104 101x2)
    Rectangle (267,108 101x24), "iPort0Pin4"
    Rectangle (267,136 101x2)
    Rectangle (267,140 101x24), "iPort1Pin2"
    Rectangle (267,168 101x2)
    Rectangle (267,172 101x24), "iPort1Pin4"
    Rectangle (267,200 101x2)
    Rectangle (267,204 101x24), "iPort2Pin2"
    Rectangle (267,232 101x2)
    Rectangle (267,236 101x24), "iPort2Pin4"
    Rectangle (267,264 101x2)
    Rectangle (267,268 101x24), "iPort3Pin2"
    Rectangle (267,296 101x2)
    Rectangle (267,300 101x24), "iPort3Pin4"
    Rectangle (267,328 101x2)
    Rectangle (267,332 101x24), "iPort4Pin2"
    Rectangle (267,360 101x2)
    Rectangle (267,364 101x24), "iPort4Pin4"
    Rectangle (267,392 101x2)
    Rectangle (267,396 101x24), "iPort5Pin2"
    Rectangle (267,424 101x2)
    Rectangle (267,428 101x24), "iPort5Pin4"
    Rectangle (267,456 101x2)
    Rectangle (267,460 101x24), "iPort6Pin2"
    Rectangle (267,488 101x2)
    Rectangle (267,492 101x24), "iPort6Pin4"
    Rectangle (267,520 101x2)
    Rectangle (267,524 101x24), "iPort7Pin2"
    Rectangle (267,552 101x2)
    Rectangle (267,556 101x24), "iPort7Pin4"
    Rectangle (267,584 101x2)
END_VISUALIZATION

// /VISU_NEW_FB_Murr56691_IP20
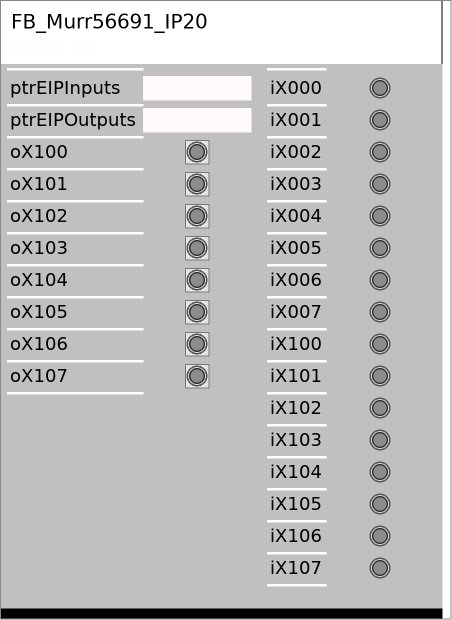
VISUALIZATION VISU_NEW_FB_Murr56691_IP20  // 452x620
VAR_INPUT
   {attribute 'parameterstringof' := 'm_Input_FB'}
   m_Input_INST_Str : STRING;
END_VAR
VAR_IN_OUT
   m_Input_FB : FB_Murr56691_IP20;
END_VAR
    RoundedRectangle (0,0 442x81)
    RoundedRectangle (0,578 442x40)
    Rectangle (0,64 442x544)
    Lamp1 (368,76 24x24), variable: m_Input_FB.iX000, style: Lamp-Lamp1-Gray
    Lamp1 (368,108 24x24), variable: m_Input_FB.iX001, style: Lamp-Lamp1-Gray
    Lamp1 (368,140 24x24), variable: m_Input_FB.iX002, style: Lamp-Lamp1-Gray
    Lamp1 (368,172 24x24), variable: m_Input_FB.iX003, style: Lamp-Lamp1-Gray
    Lamp1 (368,204 24x24), variable: m_Input_FB.iX004, style: Lamp-Lamp1-Gray
    Lamp1 (368,236 24x24), variable: m_Input_FB.iX005, style: Lamp-Lamp1-Gray
    Lamp1 (368,268 24x24), variable: m_Input_FB.iX006, style: Lamp-Lamp1-Gray
    Lamp1 (368,300 24x24), variable: m_Input_FB.iX007, style: Lamp-Lamp1-Gray
    Lamp1 (368,332 24x24), variable: m_Input_FB.iX100, style: Lamp-Lamp1-Gray
    Lamp1 (368,364 24x24), variable: m_Input_FB.iX101, style: Lamp-Lamp1-Gray
    Lamp1 (368,396 24x24), variable: m_Input_FB.iX102, style: Lamp-Lamp1-Gray
    Lamp1 (368,428 24x24), variable: m_Input_FB.iX103, style: Lamp-Lamp1-Gray
    Lamp1 (368,460 24x24), variable: m_Input_FB.iX104, style: Lamp-Lamp1-Gray
    Lamp1 (368,492 24x24), variable: m_Input_FB.iX105, style: Lamp-Lamp1-Gray
    Lamp1 (368,524 24x24), variable: m_Input_FB.iX106, style: Lamp-Lamp1-Gray
    Lamp1 (368,556 24x24), variable: m_Input_FB.iX107, style: Lamp-Lamp1-Gray
    PushSwitch (185,140 24x24), variable: m_Input_FB.oX100, behaviour: TOGGLE, style: Switch-PushSwitch-Gray
    PushSwitch (185,172 24x24), variable: m_Input_FB.oX101, behaviour: TOGGLE, style: Switch-PushSwitch-Gray
    PushSwitch (185,204 24x24), variable: m_Input_FB.oX102, behaviour: TOGGLE, style: Switch-PushSwitch-Gray
    PushSwitch (185,236 24x24), variable: m_Input_FB.oX103, behaviour: TOGGLE, style: Switch-PushSwitch-Gray
    PushSwitch (185,268 24x24), variable: m_Input_FB.oX104, behaviour: TOGGLE, style: Switch-PushSwitch-Gray
    PushSwitch (185,300 24x24), variable: m_Input_FB.oX105, behaviour: TOGGLE, style: Switch-PushSwitch-Gray
    PushSwitch (185,332 24x24), variable: m_Input_FB.oX106, behaviour: TOGGLE, style: Switch-PushSwitch-Gray
    PushSwitch (185,364 24x24), variable: m_Input_FB.oX107, behaviour: TOGGLE, style: Switch-PushSwitch-Gray
    Rectangle (8,8 442x27), "FB_Murr56691_IP20"
    Rectangle (8,35 442x27), "Instance: %s", text variable: m_Input_INST_Str
    Rectangle (7,68 136x2)
    Rectangle (143,76 108x24), text variable: m_Input_FB.ptrEIPInputs
        OnMouseClick: write the text variable via Default
    Rectangle (7,76 136x24), "ptrEIPInputs"
    Rectangle (7,104 136x2)
    Rectangle (143,108 108x24), text variable: m_Input_FB.ptrEIPOutputs
        OnMouseClick: write the text variable via Default
    Rectangle (7,108 136x24), "ptrEIPOutputs"
    Rectangle (7,136 136x2)
    Rectangle (7,140 136x24), "oX100"
    Rectangle (7,168 136x2)
    Rectangle (7,172 136x24), "oX101"
    Rectangle (7,200 136x2)
    Rectangle (7,204 136x24), "oX102"
    Rectangle (7,232 136x2)
    Rectangle (7,236 136x24), "oX103"
    Rectangle (7,264 136x2)
    Rectangle (7,268 136x24), "oX104"
    Rectangle (7,296 136x2)
    Rectangle (7,300 136x24), "oX105"
    Rectangle (7,328 136x2)
    Rectangle (7,332 136x24), "oX106"
    Rectangle (7,360 136x2)
    Rectangle (7,364 136x24), "oX107"
    Rectangle (7,392 136x2)
    Rectangle (267,68 59x2)
    Rectangle (267,76 59x24), "iX000"
    Rectangle (267,104 59x2)
    Rectangle (267,108 59x24), "iX001"
    Rectangle (267,136 59x2)
    Rectangle (267,140 59x24), "iX002"
    Rectangle (267,168 59x2)
    Rectangle (267,172 59x24), "iX003"
    Rectangle (267,200 59x2)
    Rectangle (267,204 59x24), "iX004"
    Rectangle (267,232 59x2)
    Rectangle (267,236 59x24), "iX005"
    Rectangle (267,264 59x2)
    Rectangle (267,268 59x24), "iX006"
    Rectangle (267,296 59x2)
    Rectangle (267,300 59x24), "iX007"
    Rectangle (267,328 59x2)
    Rectangle (267,332 59x24), "iX100"
    Rectangle (267,360 59x2)
    Rectangle (267,364 59x24), "iX101"
    Rectangle (267,392 59x2)
    Rectangle (267,396 59x24), "iX102"
    Rectangle (267,424 59x2)
    Rectangle (267,428 59x24), "iX103"
    Rectangle (267,456 59x2)
    Rectangle (267,460 59x24), "iX104"
    Rectangle (267,488 59x2)
    Rectangle (267,492 59x24), "iX105"
    Rectangle (267,520 59x2)
    Rectangle (267,524 59x24), "iX106"
    Rectangle (267,552 59x2)
    Rectangle (267,556 59x24), "iX107"
    Rectangle (267,584 59x2)
END_VISUALIZATION

// /VISU_NEW_FB_PneuBagOpenFingersWithSensors
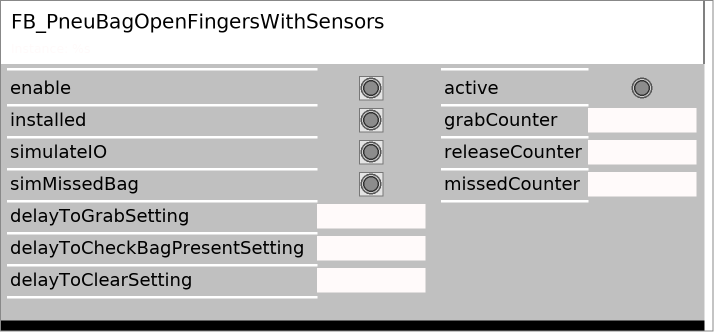
VISUALIZATION VISU_NEW_FB_PneuBagOpenFingersWithSensors  // 714x332
VAR_INPUT
   {attribute 'parameterstringof' := 'm_Input_FB'}
   m_Input_INST_Str : STRING;
END_VAR
VAR_IN_OUT
   m_Input_FB : FB_PneuBagOpenFingersWithSensorsOLD;
END_VAR
    RoundedRectangle (0,0 704x81)
    RoundedRectangle (0,290 704x40)
    Rectangle (0,64 704x256)
    Lamp1 (630,76 24x24), variable: m_Input_FB._optionActive, style: Lamp-Lamp1-Gray
    PushSwitch (359,76 24x24), variable: m_Input_FB.enable, behaviour: TOGGLE, style: Switch-PushSwitch-Gray
    PushSwitch (359,108 24x24), variable: m_Input_FB.installed, behaviour: TOGGLE, style: Switch-PushSwitch-Gray
    PushSwitch (359,140 24x24), variable: m_Input_FB.simulateIO, behaviour: TOGGLE, style: Switch-PushSwitch-Gray
    PushSwitch (359,172 24x24), variable: m_Input_FB.simMissedBag, behaviour: TOGGLE, style: Switch-PushSwitch-Gray
    Rectangle (8,8 704x27), "FB_PneuBagOpenFingersWithSensors"
    Rectangle (8,35 704x27), "Instance: %s", text variable: m_Input_INST_Str
    Rectangle (7,68 310x2)
    Rectangle (7,76 310x24), "enable"
    Rectangle (7,104 310x2)
    Rectangle (7,108 310x24), "installed"
    Rectangle (7,136 310x2)
    Rectangle (441,68 147x2)
    Rectangle (441,76 147x24), "active"
    Rectangle (441,104 147x2)
    Rectangle (7,140 310x24), "simulateIO"
    Rectangle (7,168 310x2)
    Rectangle (7,172 310x24), "simMissedBag"
    Rectangle (7,200 310x2)
    Rectangle (317,204 108x24), text variable: m_Input_FB.delayToGrabSetting
        OnMouseClick: write the text variable via Default
    Rectangle (7,204 310x24), "delayToGrabSetting"
    Rectangle (7,232 310x2)
    Rectangle (317,236 108x24), text variable: m_Input_FB.delayToCheckBagPresentSetting
        OnMouseClick: write the text variable via Default
    Rectangle (7,236 310x24), "delayToCheckBagPresentSetting"
    Rectangle (7,264 310x2)
    Rectangle (317,268 108x24), text variable: m_Input_FB.delayToClearSetting
        OnMouseClick: write the text variable via Default
    Rectangle (7,268 310x24), "delayToClearSetting"
    Rectangle (7,296 310x2)
    Rectangle (588,108 108x24), text variable: m_Input_FB.grabCounter
    Rectangle (441,108 147x24), "grabCounter"
    Rectangle (441,136 147x2)
    Rectangle (588,140 108x24), text variable: m_Input_FB.releaseCounter
    Rectangle (441,140 147x24), "releaseCounter"
    Rectangle (441,168 147x2)
    Rectangle (588,172 108x24), text variable: m_Input_FB.missedCounter
    Rectangle (441,172 147x24), "missedCounter"
    Rectangle (441,200 147x2)
END_VISUALIZATION

// /VISU_NEW_FB_PneuBagOpenFingersWithSensorsOLD
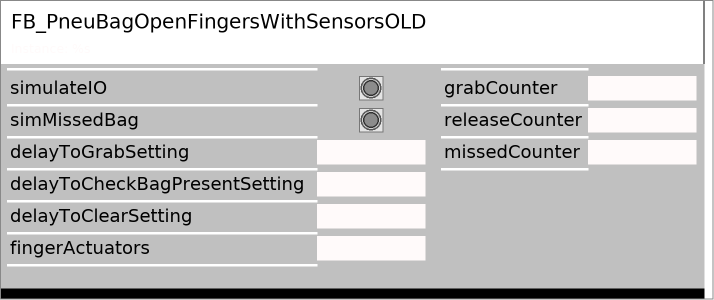
VISUALIZATION VISU_NEW_FB_PneuBagOpenFingersWithSensorsOLD  // 714x300
VAR_INPUT
   {attribute 'parameterstringof' := 'm_Input_FB'}
   m_Input_INST_Str : STRING;
END_VAR
VAR_IN_OUT
   m_Input_FB : FB_PneuBagOpenFingersWithSensorsOLD;
END_VAR
    RoundedRectangle (0,0 704x81)
    RoundedRectangle (0,258 704x40)
    Rectangle (0,64 704x224)
    PushSwitch (359,76 24x24), variable: m_Input_FB.simulateIO, behaviour: TOGGLE, style: Switch-PushSwitch-Gray
    PushSwitch (359,108 24x24), variable: m_Input_FB.simMissedBag, behaviour: TOGGLE, style: Switch-PushSwitch-Gray
    Rectangle (8,8 704x27), "FB_PneuBagOpenFingersWithSensorsOLD"
    Rectangle (8,35 704x27), "Instance: %s", text variable: m_Input_INST_Str
    Rectangle (7,68 310x2)
    Rectangle (7,76 310x24), "simulateIO"
    Rectangle (7,104 310x2)
    Rectangle (7,108 310x24), "simMissedBag"
    Rectangle (7,136 310x2)
    Rectangle (317,140 108x24), text variable: m_Input_FB.delayToGrabSetting
        OnMouseClick: write the text variable via Default
    Rectangle (7,140 310x24), "delayToGrabSetting"
    Rectangle (7,168 310x2)
    Rectangle (317,172 108x24), text variable: m_Input_FB.delayToCheckBagPresentSetting
        OnMouseClick: write the text variable via Default
    Rectangle (7,172 310x24), "delayToCheckBagPresentSetting"
    Rectangle (7,200 310x2)
    Rectangle (317,204 108x24), text variable: m_Input_FB.delayToClearSetting
        OnMouseClick: write the text variable via Default
    Rectangle (7,204 310x24), "delayToClearSetting"
    Rectangle (7,232 310x2)
    Rectangle (441,68 147x2)
    Rectangle (588,76 108x24), text variable: m_Input_FB.grabCounter
    Rectangle (441,76 147x24), "grabCounter"
    Rectangle (441,104 147x2)
    Rectangle (588,108 108x24), text variable: m_Input_FB.releaseCounter
    Rectangle (441,108 147x24), "releaseCounter"
    Rectangle (441,136 147x2)
    Rectangle (588,140 108x24), text variable: m_Input_FB.missedCounter
    Rectangle (441,140 147x24), "missedCounter"
    Rectangle (441,168 147x2)
    Rectangle (317,236 108x24), text variable: m_Input_FB.fingerActuators
        OnMouseClick: write the text variable via Default
    Rectangle (7,236 310x24), "fingerActuators"
    Rectangle (7,264 310x2)
END_VISUALIZATION

// /VISU_NEW_FB_Simulation
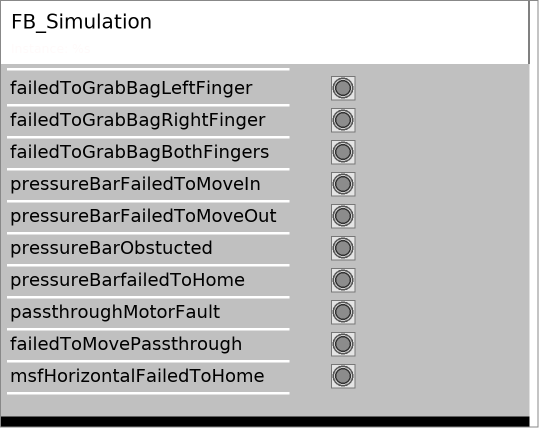
VISUALIZATION VISU_NEW_FB_Simulation  // 539x428
VAR_INPUT
   {attribute 'parameterstringof' := 'm_Input_FB'}
   m_Input_INST_Str : STRING;
END_VAR
VAR_IN_OUT
   m_Input_FB : FB_Simulation;
END_VAR
    RoundedRectangle (0,0 529x81)
    RoundedRectangle (0,386 529x40)
    Rectangle (0,64 529x352)
    PushSwitch (331,76 24x24), variable: m_Input_FB.failedToGrabBagLeftFinger, behaviour: TOGGLE, style: Switch-PushSwitch-Gray
    PushSwitch (331,108 24x24), variable: m_Input_FB.failedToGrabBagRightFinger, behaviour: TOGGLE, style: Switch-PushSwitch-Gray
    PushSwitch (331,140 24x24), variable: m_Input_FB.failedToGrabBagBothFingers, behaviour: TOGGLE, style: Switch-PushSwitch-Gray
    PushSwitch (331,172 24x24), variable: m_Input_FB.pressureBarFailedToMoveIn, behaviour: TOGGLE, style: Switch-PushSwitch-Gray
    PushSwitch (331,204 24x24), variable: m_Input_FB.pressureBarFailedToMoveOut, behaviour: TOGGLE, style: Switch-PushSwitch-Gray
    PushSwitch (331,236 24x24), variable: m_Input_FB.pressureBarObstucted, behaviour: TOGGLE, style: Switch-PushSwitch-Gray
    PushSwitch (331,268 24x24), variable: m_Input_FB.pressureBarfailedToHome, behaviour: TOGGLE, style: Switch-PushSwitch-Gray
    PushSwitch (331,300 24x24), variable: m_Input_FB.passthroughMotorFault, behaviour: TOGGLE, style: Switch-PushSwitch-Gray
    PushSwitch (331,332 24x24), variable: m_Input_FB.failedToMovePassthrough, behaviour: TOGGLE, style: Switch-PushSwitch-Gray
    PushSwitch (331,364 24x24), variable: m_Input_FB.msfHorizontalFailedToHome, behaviour: TOGGLE, style: Switch-PushSwitch-Gray
    Rectangle (8,8 529x27), "FB_Simulation"
    Rectangle (8,35 529x27), "Instance: %s", text variable: m_Input_INST_Str
    Rectangle (7,68 282x2)
    Rectangle (7,76 282x24), "failedToGrabBagLeftFinger"
    Rectangle (7,104 282x2)
    Rectangle (7,108 282x24), "failedToGrabBagRightFinger"
    Rectangle (7,136 282x2)
    Rectangle (7,140 282x24), "failedToGrabBagBothFingers"
    Rectangle (7,168 282x2)
    Rectangle (7,172 282x24), "pressureBarFailedToMoveIn"
    Rectangle (7,200 282x2)
    Rectangle (7,204 282x24), "pressureBarFailedToMoveOut"
    Rectangle (7,232 282x2)
    Rectangle (7,236 282x24), "pressureBarObstucted"
    Rectangle (7,264 282x2)
    Rectangle (7,268 282x24), "pressureBarfailedToHome"
    Rectangle (7,296 282x2)
    Rectangle (7,300 282x24), "passthroughMotorFault"
    Rectangle (7,328 282x2)
    Rectangle (7,332 282x24), "failedToMovePassthrough"
    Rectangle (7,360 282x2)
    Rectangle (7,364 282x24), "msfHorizontalFailedToHome"
    Rectangle (7,392 282x2)
END_VISUALIZATION

// UN00 - Sharp Bagger/PackML
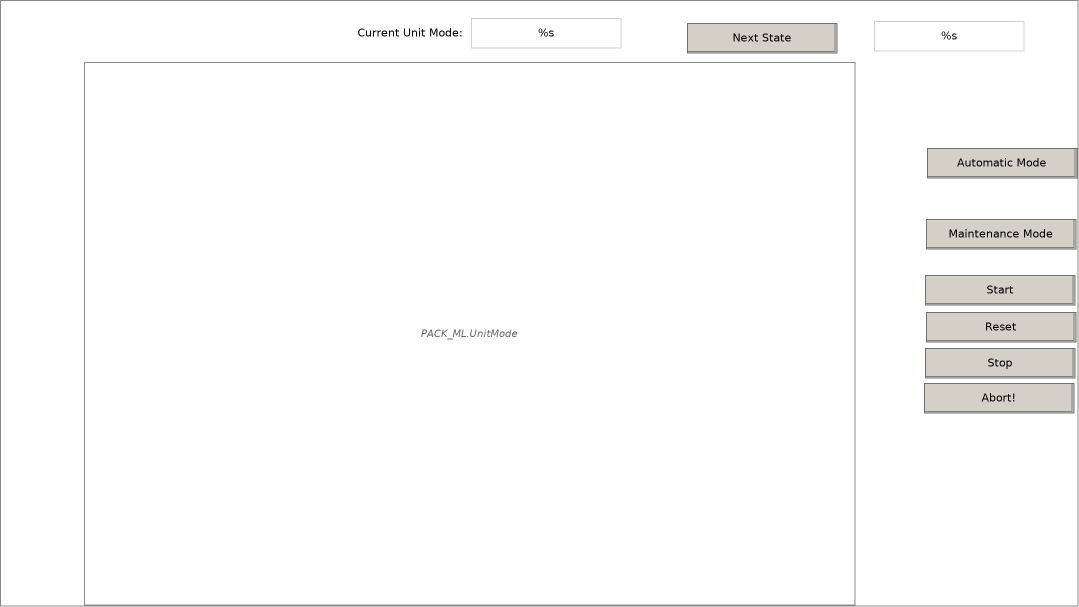
VISUALIZATION PackML  // 1079x607
VAR_IN_OUT
	Machine : FB_UN00_SharpMachine;
END_VAR
    Frame (84,62 771x543)
        shows PACK_ML.UnitMode(um := Machine.currentUnitMode)
    Label (335,18 150x30), "Current Unit Mode:"
    Textfield (471,18 150x30), "%s", text variable: Machine.sCurrentUnitModeName
    Button (927,148 150x30), "Automatic Mode"
        OnMouseDown: execute { Machine.unitModeManager.SwitchUnitMode(UN00_Globals.sAutomatic); }
    Button (926,219 150x30), "Maintenance Mode"
        OnMouseDown: execute { Machine.unitModeManager.SwitchUnitMode(UN00_Globals.sMaintenance); }
    Button (687,23 150x30), "Next State"
        OnMouseDown:  ToggleVariable=Machine.xNextState
    Textfield (874,21 150x30), "%s", text variable: Machine.currentState
    Button (924,383 150x30), "Abort!"
        OnMouseClick:  ToggleVariable=Machine.abortMachine
    Button (926,312 150x30), "Reset"
        tap Machine.resetMachine
    Button (925,275 150x30), "Start"
        OnMouseClick:  ToggleVariable=Machine.startMachine
    Button (925,348 150x30), "Stop"
        OnMouseClick: execute { Machine.currentUnitMode.Stop(); }
END_VISUALIZATION

(* text list System (id | default)
  Apr | Apr
  April | April
  Aug | Aug
  August | August
  Dec | Dec
  December | December
  Feb | Feb
  February | February
  Fri | Fri
  Friday | Friday
  Jan | Jan
  January | January
  Jul | Jul
  July | July
  Jun | Jun
  June | June
  Mar | Mar
  March | March
  May | May
  May_3Letter | May
  Mon | Mon
  Monday | Monday
  Nov | Nov
  November | November
  Oct | Oct
  October | October
  Sat | Sat
  Saturday | Saturday
  Sep | Sep
  September | September
  Sun | Sun
  Sunday | Sunday
  Thu | Thu
  Thursday | Thursday
  Tue | Tue
  Tuesday | Tuesday
  Wed | Wed
  Wednesday | Wednesday
   |  *)

(* text list TextListForCombobox_BagOpenFingersSelection (id | default)
  0 | NOTINSTALLED
  1 | PNEUMATICWITHBAGOPENSENSORS
   |  *)

(* text list TextListForCombobox_IntegratedConveyorSelection (id | default)
  0 | NOTINSTALLED
  1 | REAREXIT
   |  *)

(* text list TextListForCombobox_LabelPrinterSelection (id | default)
  0 | NOTINSTALLED
  1 | ZEBRAPRINTER
   |  *)

(* text list TextListForCombobox_PackageEjectionSelection (id | default)
  0 | NOTINSTALLED
  1 | REARRETRACTINGLOADPLATE
  2 | LABELSIDEUP
   |  *)

(* text list TextListForCombobox_SealFlattenerSelection (id | default)
  0 | NOTINSTALLED
  1 | MOTORIZEDSEALFLATTENERS
   |  *)
